Staubli VAL3: SplitChar.pgx

public program SplitChar(num& x_nRes, string x_sStrIn, string x_sChar, string& x_sOut[])
  local string l_sBuff
  local num l_nIndex
  local num l_nLen
  local num l_nCharLen
  local num l_nStrIndex
begin
  //****************************************************************
  //***************************************************************
  //函数名称：SplitChar
  //用途：  用于解析字符
  //创建日期：
  //作者：
  //联系方式：
  //备注：
  //版本修改说明：
  //****************************************************************
  //*****************************************************************
  //1.参数定义
  l_sBuff=""
  l_nIndex=0
  l_nLen=0
  while size(x_sOut)>1
    delete(x_sOut[0])
  endWhile
  x_sOut[0]=""

  //2.条件判断
  if x_sStrIn=="" or x_sChar==""
    x_nRes=-1
    return
  endIf
  l_nCharLen=len(x_sChar)

  //3.分割字符串
  while find(x_sStrIn,x_sChar)>=0
    l_nStrIndex=find(x_sStrIn,x_sChar)
    l_nLen=l_nCharLen+l_nStrIndex
    x_sOut[l_nIndex]=left(x_sStrIn,l_nStrIndex)
    l_nIndex=l_nIndex+1
    insert(x_sOut[l_nIndex])
    x_sStrIn=delete(x_sStrIn,l_nLen,0)
  endWhile
  if x_sStrIn!=""
    x_sOut[l_nIndex]=x_sStrIn
  else
    delete(x_sOut[l_nIndex])
  endIf
  x_nRes=0
end
